FUNCTION_BLOCK FB_TBlink
VAR_INPUT
	IN: BOOL;
	PT: TIME;
END_VAR
VAR_OUTPUT
	Q: BOOL;
END_VAR
VAR
	fbTimer: TP;
END_VAR

fbTimer(IN:=IN AND NOT fbTimer.Q, PT:=PT);

IF IN AND fbTimer.ET < PT/2 THEN
	Q := TRUE;
ELSE
	Q := FALSE;
END_IF

END_FUNCTION_BLOCK

(* stored: Version 1.1.0.1, ProductVersion 3.1.4024.3
   POU FB_TBlink: Id {b73d6dc6-f70e-406e-8d5b-e7b4e5f0b150}, SpecialFunc None *)
